(* PLC project Unnamed, Unknown Unnamed 1 *)
(* stored: creationDateTime 2026-02-24T10:36:00, modificationDateTime 2026-02-24T10:48:31 *)

PROGRAM program0
  VAR
    Trigger : BOOL;
    Lamp : BOOL;
    TON0 : TON;
    TOF0 : TOF;
  END_VAR

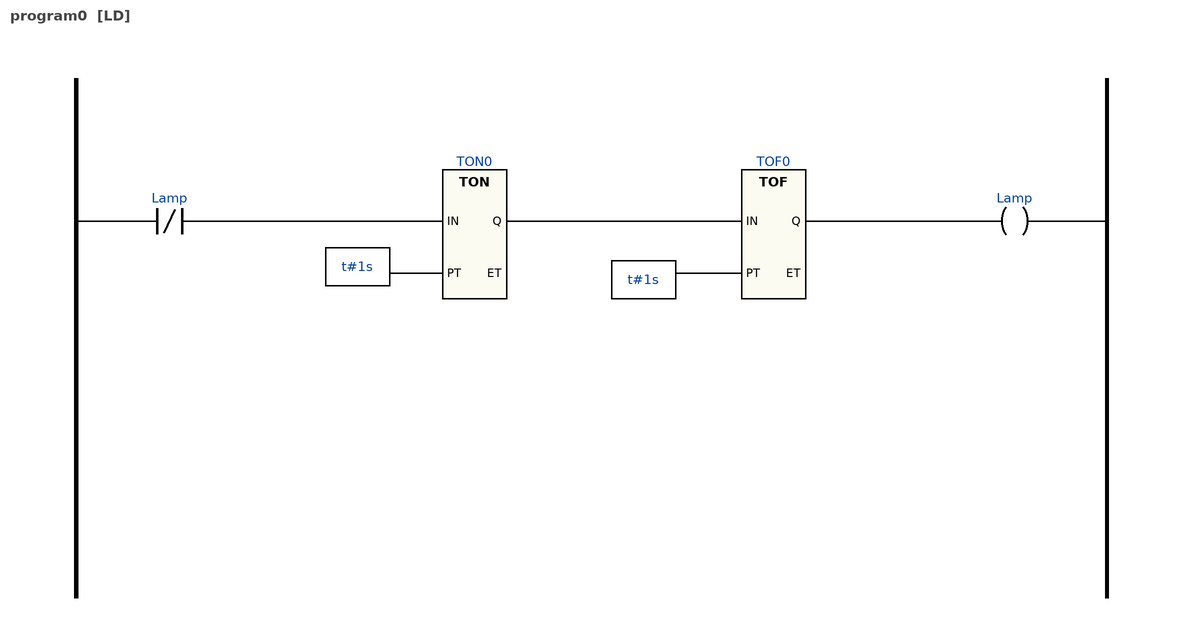
(* LD diagram, written out as Structured Text *)
TON0(IN := NOT Lamp, PT := t#1s);
TOF0(IN := TON0.Q, PT := t#1s);
Lamp := TOF0.Q;
END_PROGRAM

CONFIGURATION Config0
  RESOURCE Res0 ON PLC
    TASK task0(INTERVAL := T#20ms, PRIORITY := 0);
    PROGRAM instance0 WITH task0 : program0;
  END_RESOURCE
END_CONFIGURATION
